FUNCTION_BLOCK StructConsumer (* Simple FB with one algorithm *)
  (* Standard: 61499-1 *)
  (* Version 1.0, 2026-06-17, Dimitrios Kalligaridis *)
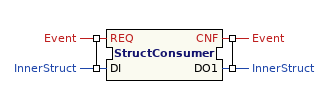
  EVENT_INPUT
    REQ WITH DI; (* Normal Execution Request *)
  END_EVENT
  EVENT_OUTPUT
    CNF WITH DO1; (* Execution Confirmation *)
  END_EVENT
  VAR_INPUT
    DI : mypackage::InnerStruct;
  END_VAR
  VAR_OUTPUT
    DO1 : mypackage::InnerStruct;
  END_VAR
  EC_STATES
    REQ : REQ -> CNF;
  END_STATES
  ALGORITHM REQ IN ST:

  END_ALGORITHM
END_FUNCTION_BLOCK
